PROGRAM TCPServer
VAR	
	bSuccess					: BOOL;//函数 F_CreateServerHnd 用于初始化句柄 hServer 内部参数并创建服务器，bSuccess确认是否建立成功
	bEnable						: BOOL;//是否启用
	Step						: INT;
	iCount						: INT;

	//控制器做 TCPIP 的 Server
	sRemoteHost 				: STRING(15) := '169.254.130.170';//控制器IP地址
	nRemotePort 				: UDINT := 2000;//控制器端口号
	fb_ServerConnection			: FB_ServerClientConnection;//建立server 和client连接
	hServer						: T_HSERVER;//TCPIP被创建的服务器
	hSocket						: T_HSOCKET;//TCPIP句柄

	//数据接收
	fb_Receive					: FB_SocketReceive;
//	Data_receive	   AT%Q*	: ARRAY[1..10]OF BYTE;
//	bReceive		   AT%I*	: BOOL;//接收执行
	
	//数据发送
	fb_Send						: FB_SocketSend;
//	nSendDataBuffer	   AT%I*	: ARRAY[1..50]OF BYTE;
//	bsend			   AT%I*	: BOOL;//发送执行
END_VAR

FBD();
CASE step OF
0:
	bSuccess:=FALSE;
    bEnable:=FALSE;
         step:=step+1;
1:
	bSuccess:=F_CreateServerHnd(
	sSrvNetID:='' ,
	sLocalHost:=sRemoteHost ,
	nLocalPort:=nRemotePort ,
	nMode:=LISTEN_MODE_CLOSEALL OR CONNECT_MODE_ENABLEDBG ,
	bEnable:=TRUE ,
	hServer:=hserver );
         step:=step+1;

2:
        IF bSuccess THEN
 	       bEnable:=TRUE;
	        IF  NOT fb_ServerConnection.bError THEN
		          step:=step+1;
	         ELSE
 		        step:=0;
   	      	END_IF
      	ELSE
	         step:=0;
      	END_IF

3:
		IF fb_ServerConnection.eState=eSOCKET_CONNECTED THEN
				iCount:=iCount+1;
 				step:=step+1;
		END_IF

4:

    fb_Receive(
	sSrvNetId:='' ,
	hSocket:=hSocket ,
	cbLen:=SIZEOF(GVL.Data_receive) ,
	pDest:=ADR(GVL.Data_receive) ,
	bExecute:=GVL.bReceive ,
	tTimeout:=T#1S ,
	bBusy=> ,
	bError=> ,
	nErrId=> ,
	nRecBytes=> );
IF   NOT fb_Receive.bbusy OR NOT fb_Receive.berror THEN
	fb_Send(
	sSrvNetId:='' ,
	hSocket:=hSocket ,
	cbLen:=SIZEOF(GVL.nSendDataBuffer) ,
	pSrc:=ADR(GVL.nSendDataBuffer) ,
	bExecute:=GVL.bsend ,
	tTimeout:=t#6s ,
	bBusy=> ,
	bError=> ,
	nErrId=> );
END_IF
//		ELSE
//   		 step:=0;
GVL.rec_busy:=fb_Receive.bBusy;
IF fb_Receive.nRecBytes>0 THEN
			GVL.number_recdata:=fb_Receive.nRecBytes;//返回接收到的数据个数
END_IF	
IF GVL.bReceive=TRUE THEN
			GVL.bReceive:=FALSE;//只接收一次数据
END_IF
IF GVL.bsend=TRUE THEN
			GVL.bsend:=FALSE;//只发送一次数据
END_IF
END_CASE

ACTION FBD:
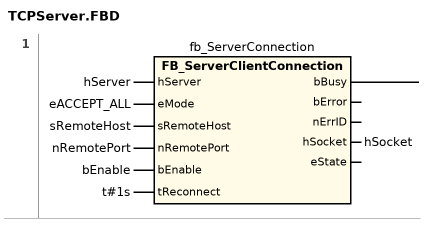
// NETWORK 1
fb_ServerConnection(
    hServer := hServer,
    eMode := eACCEPT_ALL,
    sRemoteHost := sRemoteHost,
    nRemotePort := nRemotePort,
    bEnable := bEnable,
    tReconnect := t#1s,
    hSocket => hSocket); // FB_ServerClientConnection
END_ACTION

END_PROGRAM

(* stored: Version 1.1.0.1, ProductVersion 3.1.4024.15
   POU TCPServer: Id {e7ca4252-f97d-44e0-bcf2-5e3d5d0e1ef7}, SpecialFunc None
   Action FBD: Id {815295f9-a16f-4cfb-afcc-ba3c47d9c10e} *)
